// TIA Portal V18 export
ORGANIZATION_BLOCK "Main"   // OB1, LAD, ProgramCycle
TITLE = "Main Program Sweep (Cycle)"
{ S7_Optimized_Access := 'TRUE' }
VERSION : 0.1
// stored: AutoNumber true, IsIECCheckEnabled false, SetENOAutomatically false
   VAR_INPUT
      Initial_Call : Bool;   // Initial call of this OB
      Remanence : Bool;   // =True, if remanent data are available
   END_VAR
   VAR_TEMP
      temp1 : Bool;
      temp2 : Bool;
      temp3 : Bool;
      temp4 : Bool;
   END_VAR
   VAR_TEMP   // added for the SCL form of the ladder/FBD networks
      _w1 : Bool;
      _w2 : Bool;
      _w3 : Bool;
      _w4 : Bool;
      _w5 : Bool;
      _w6 : Bool;
      _w7 : Bool;
      _w8 : Bool;
      _w9 : Bool;
      _w10 : Bool;
      _w11 : Bool;
      _w12 : Bool;
      _w13 : Bool;
      _w14 : Bool;
      _w15 : Bool;
      _w16 : Bool;
   END_VAR
BEGIN

REGION Network 1: SFC1
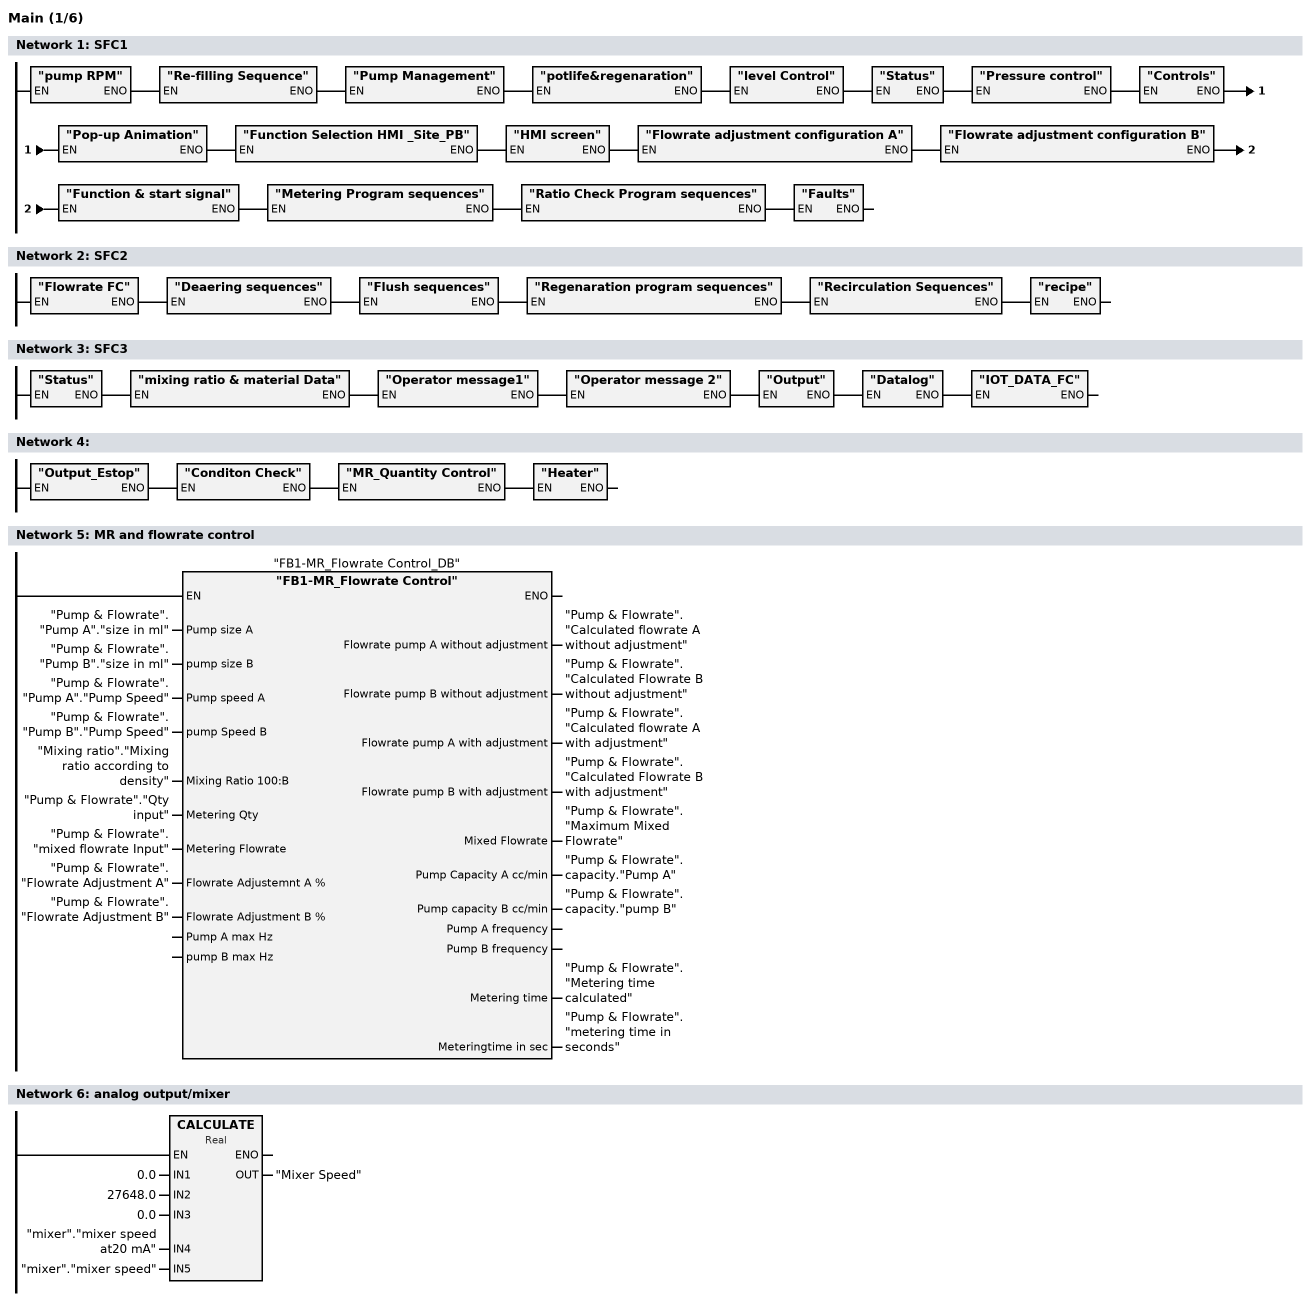
   RUNG wire#powerrail
      "pump RPM"()
      "Re-filling Sequence"()
      "Pump Management"()
      "potlife&regenaration"()
      "level Control"()
      "Status"()
      "Pressure control"()
      "Controls"()
      "Pop-up Animation"()
      "Function Selection HMI _Site_PB"()
      "HMI screen"()
      "Flowrate adjustment configuration A"()
      "Flowrate adjustment configuration B"()
      "Function & start signal"()
      "Metering Program sequences"()
      "Ratio Check Program sequences"()
      "Faults"()
   END_RUNG
   // the same network as SCL:
   "pump RPM"(ENO => #_w1);
   "Re-filling Sequence"(EN := #_w1, ENO => #_w2);
   "Pump Management"(EN := #_w2, ENO => #_w3);
   "potlife&regenaration"(EN := #_w3, ENO => #_w4);
   "level Control"(EN := #_w4, ENO => #_w5);
   "Status"(EN := #_w5, ENO => #_w6);
   "Pressure control"(EN := #_w6, ENO => #_w7);
   "Controls"(EN := #_w7, ENO => #_w8);
   "Pop-up Animation"(EN := #_w8, ENO => #_w9);
   "Function Selection HMI _Site_PB"(EN := #_w9, ENO => #_w10);
   "HMI screen"(EN := #_w10, ENO => #_w11);
   "Flowrate adjustment configuration A"(EN := #_w11, ENO => #_w12);
   "Flowrate adjustment configuration B"(EN := #_w12, ENO => #_w13);
   "Function & start signal"(EN := #_w13, ENO => #_w14);
   "Metering Program sequences"(EN := #_w14, ENO => #_w15);
   "Ratio Check Program sequences"(EN := #_w15, ENO => #_w16);
   IF #_w16 THEN "Faults"(); END_IF;
END_REGION

REGION Network 2: SFC2
   RUNG wire#powerrail
      "Flowrate FC"()
      "Deaering sequences"()
      "Flush sequences"()
      "Regenaration program sequences"()
      "Recirculation Sequences"()
      "recipe"()
   END_RUNG
   // the same network as SCL:
   "Flowrate FC"(ENO => #_w1);
   "Deaering sequences"(EN := #_w1, ENO => #_w2);
   "Flush sequences"(EN := #_w2, ENO => #_w3);
   "Regenaration program sequences"(EN := #_w3, ENO => #_w4);
   "Recirculation Sequences"(EN := #_w4, ENO => #_w5);
   IF #_w5 THEN "recipe"(); END_IF;
END_REGION

REGION Network 3: SFC3
   RUNG wire#powerrail
      "Status"()
      "mixing ratio & material Data"()
      "Operator message1"()
      "Operator message 2"()
      "Output"()
      "Datalog"()
      "IOT_DATA_FC"()
   END_RUNG
   // the same network as SCL:
   "Status"(ENO => #_w1);
   "mixing ratio & material Data"(EN := #_w1, ENO => #_w2);
   "Operator message1"(EN := #_w2, ENO => #_w3);
   "Operator message 2"(EN := #_w3, ENO => #_w4);
   "Output"(EN := #_w4, ENO => #_w5);
   "Datalog"(EN := #_w5, ENO => #_w6);
   IF #_w6 THEN "IOT_DATA_FC"(); END_IF;
END_REGION

REGION Network 4
   RUNG wire#powerrail
      "Output_Estop"()
      "Conditon Check"()
      "MR_Quantity Control"()
      "Heater"()
   END_RUNG
   // the same network as SCL:
   "Output_Estop"(ENO => #_w1);
   "Conditon Check"(EN := #_w1, ENO => #_w2);
   "MR_Quantity Control"(EN := #_w2, ENO => #_w3);
   IF #_w3 THEN "Heater"(); END_IF;
END_REGION

REGION Network 5: MR and flowrate control
   "FB1-MR_Flowrate Control_DB"("Pump size A" := "Pump & Flowrate"."Pump A"."size in ml",   // "FB1-MR_Flowrate Control"
                           "pump size B" := "Pump & Flowrate"."Pump B"."size in ml",
                           "Pump speed A" := "Pump & Flowrate"."Pump A"."Pump Speed",
                           "pump Speed B" := "Pump & Flowrate"."Pump B"."Pump Speed",
                           "Mixing Ratio 100:B" := "Mixing ratio"."Mixing ratio according to density",
                           "Metering Qty" := "Pump & Flowrate"."Qty input",
                           "Metering Flowrate" := "Pump & Flowrate"."mixed flowrate Input",
                           "Flowrate Adjustemnt A %" := "Pump & Flowrate"."Flowrate Adjustment A",
                           "Flowrate Adjustment B %" := "Pump & Flowrate"."Flowrate Adjustment B",
                           "Flowrate pump A without adjustment" => "Pump & Flowrate"."Calculated flowrate A without adjustment",
                           "Flowrate pump B without adjustment" => "Pump & Flowrate"."Calculated Flowrate B without adjustment",
                           "Flowrate pump A with adjustment" => "Pump & Flowrate"."Calculated flowrate A with adjustment",
                           "Flowrate pump B with adjustment" => "Pump & Flowrate"."Calculated Flowrate B  with adjustment",
                           "Mixed Flowrate" => "Pump & Flowrate"."Maximum Mixed Flowrate",
                           "Pump Capacity A cc/min" => "Pump & Flowrate".capacity."Pump A",
                           "Pump capacity B cc/min" => "Pump & Flowrate".capacity."pump B",
                           "Metering time" => "Pump & Flowrate"."Metering time calculated",
                           "Meteringtime in sec" => "Pump & Flowrate"."metering time in seconds");
END_REGION

REGION Network 6: analog output/mixer
   RUNG wire#powerrail
      { S7_Templates := "SrcType := Real"; S7_Expression := "(IN2-IN1)*(IN5-IN3)/(IN4-IN3)+IN1" } Calculate(in1 := 0.0, in2 := 27648.0, in3 := 0.0, in4 := "mixer"."mixer speed at20 mA", in5 := "mixer"."mixer speed", out => "Mixer Speed")
   END_RUNG
   // the same network as SCL:
   "Mixer Speed" := (27648.0-0.0)*("mixer"."mixer speed"-0.0)/("mixer"."mixer speed at20 mA"-0.0)+0.0;
END_REGION

REGION Network 7: Pump A Analog output without PID
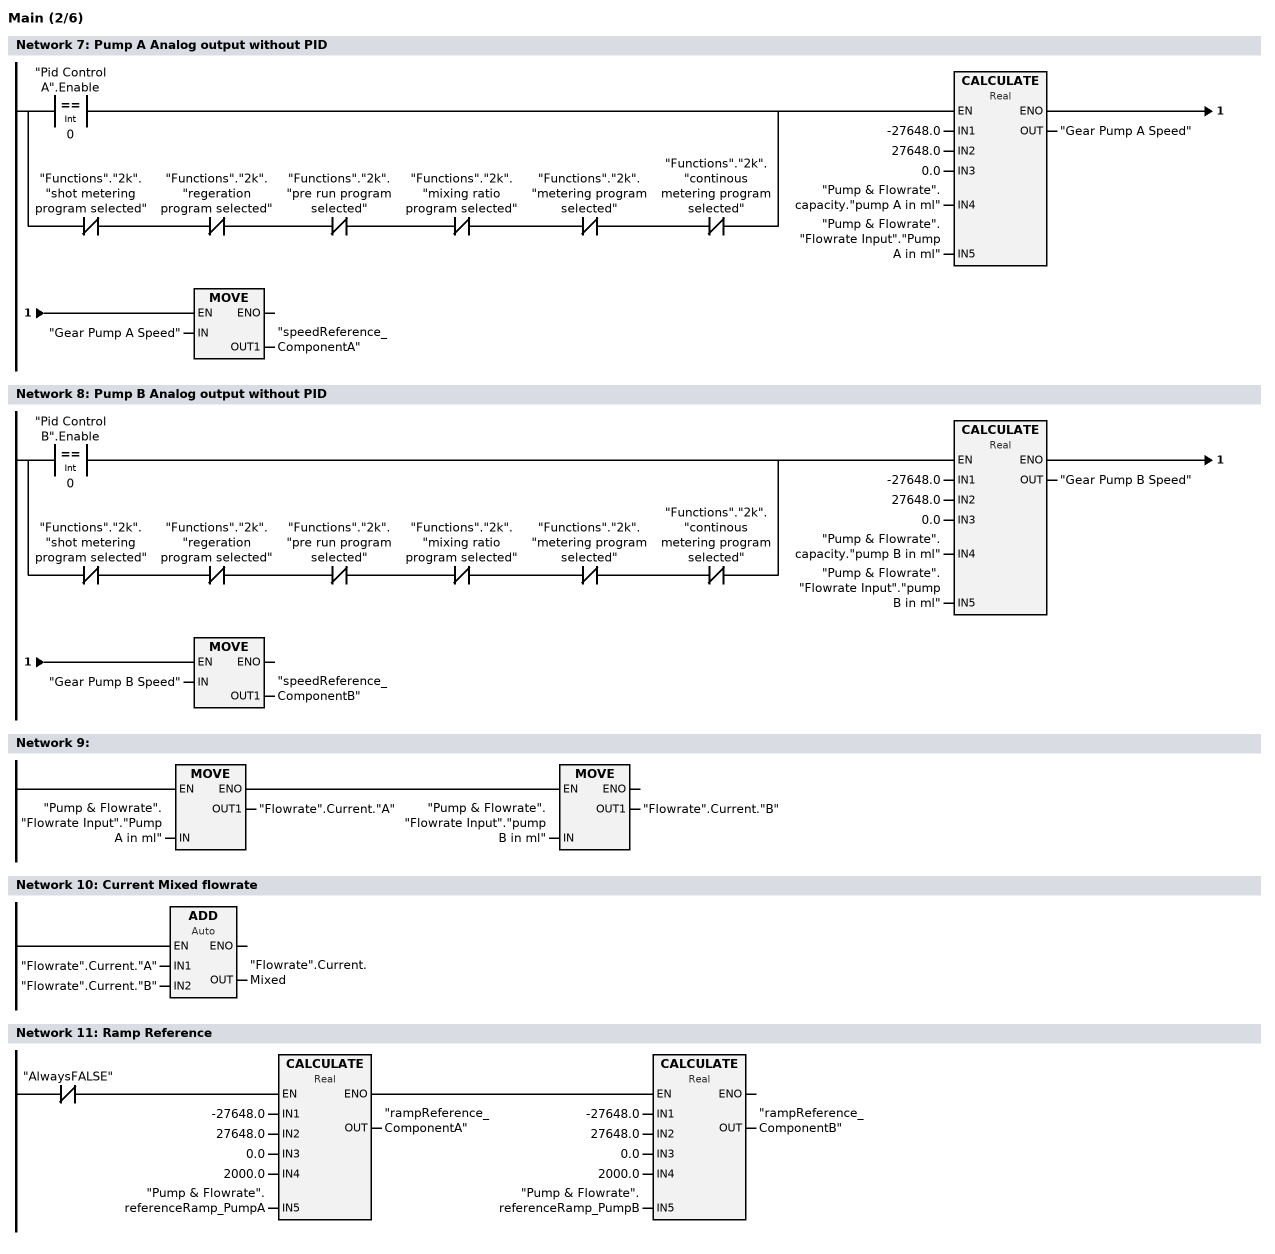
   RUNG wire#powerrail
      { S7_Templates := "SrcType := Int" } EQ_Contact(in1 := "Pid Control A".Enable, in2 := 0)
      wire#w1
      { S7_Templates := "SrcType := Real"; S7_Expression := "(IN2-IN1)*(IN5-IN3)/(IN4-IN3)+IN1" } Calculate(in1 := -27648.0, in2 := 27648.0, in3 := 0.0, in4 := "Pump & Flowrate".capacity."pump A in ml", in5 := "Pump & Flowrate"."Flowrate Input"."Pump A in ml", out => "Gear Pump A Speed")
      Move(in := "Gear Pump A Speed", out1 => "speedReference_ComponentA")
   END_RUNG
   RUNG wire#powerrail
      I_Contact( "Functions"."2k"."shot metering program selected" )
      I_Contact( "Functions"."2k"."regeration program selected" )
      I_Contact( "Functions"."2k"."pre run program selected" )
      I_Contact( "Functions"."2k"."mixing ratio program selected" )
      I_Contact( "Functions"."2k"."metering program selected" )
      I_Contact( "Functions"."2k"."continous metering program selected" )
   END_RUNG wire#w1
   // the same network as SCL:
   IF ("Pid Control A".Enable = 0) OR (NOT "Functions"."2k"."shot metering program selected" AND NOT "Functions"."2k"."regeration program selected" AND NOT "Functions"."2k"."pre run program selected" AND NOT "Functions"."2k"."mixing ratio program selected" AND NOT "Functions"."2k"."metering program selected" AND NOT "Functions"."2k"."continous metering program selected") THEN
       "Gear Pump A Speed" := (27648.0-(-27648.0))*("Pump & Flowrate"."Flowrate Input"."Pump A in ml"-0.0)/("Pump & Flowrate".capacity."pump A in ml"-0.0)+(-27648.0);
       "speedReference_ComponentA" := "Gear Pump A Speed";
   END_IF;
END_REGION

REGION Network 8: Pump B Analog output without PID
   RUNG wire#powerrail
      { S7_Templates := "SrcType := Int" } EQ_Contact(in1 := "Pid Control B".Enable, in2 := 0)
      wire#w1
      { S7_Templates := "SrcType := Real"; S7_Expression := "(IN2-IN1)*(IN5-IN3)/(IN4-IN3)+IN1" } Calculate(in1 := -27648.0, in2 := 27648.0, in3 := 0.0, in4 := "Pump & Flowrate".capacity."pump B in ml", in5 := "Pump & Flowrate"."Flowrate Input"."pump B in ml", out => "Gear Pump B Speed")
      Move(in := "Gear Pump B Speed", out1 => "speedReference_ComponentB")
   END_RUNG
   RUNG wire#powerrail
      I_Contact( "Functions"."2k"."shot metering program selected" )
      I_Contact( "Functions"."2k"."regeration program selected" )
      I_Contact( "Functions"."2k"."pre run program selected" )
      I_Contact( "Functions"."2k"."mixing ratio program selected" )
      I_Contact( "Functions"."2k"."metering program selected" )
      I_Contact( "Functions"."2k"."continous metering program selected" )
   END_RUNG wire#w1
   // the same network as SCL:
   IF ("Pid Control B".Enable = 0) OR (NOT "Functions"."2k"."shot metering program selected" AND NOT "Functions"."2k"."regeration program selected" AND NOT "Functions"."2k"."pre run program selected" AND NOT "Functions"."2k"."mixing ratio program selected" AND NOT "Functions"."2k"."metering program selected" AND NOT "Functions"."2k"."continous metering program selected") THEN
       "Gear Pump B Speed" := (27648.0-(-27648.0))*("Pump & Flowrate"."Flowrate Input"."pump B in ml"-0.0)/("Pump & Flowrate".capacity."pump B in ml"-0.0)+(-27648.0);
       "speedReference_ComponentB" := "Gear Pump B Speed";
   END_IF;
END_REGION

REGION Network 9
   RUNG wire#powerrail
      Move(in := "Pump & Flowrate"."Flowrate Input"."Pump A in ml", out1 => "Flowrate".Current."A")
      Move(in := "Pump & Flowrate"."Flowrate Input"."pump B in ml", out1 => "Flowrate".Current."B")
   END_RUNG
   // the same network as SCL:
   "Flowrate".Current."A" := "Pump & Flowrate"."Flowrate Input"."Pump A in ml";
   "Flowrate".Current."B" := "Pump & Flowrate"."Flowrate Input"."pump B in ml";
END_REGION

REGION Network 10: Current Mixed flowrate
   RUNG wire#powerrail
      Add(in1 := "Flowrate".Current."A", in2 := "Flowrate".Current."B", out => "Flowrate".Current.Mixed)
   END_RUNG
   // the same network as SCL:
   "Flowrate".Current.Mixed := "Flowrate".Current."A" + "Flowrate".Current."B";
END_REGION

REGION Network 11: Ramp Reference
   RUNG wire#powerrail
      I_Contact( "AlwaysFALSE" )
      { S7_Templates := "SrcType := Real"; S7_Expression := "ROUND((IN2-IN1)*(IN5-IN3)/(IN4-IN3)+IN1)" } Calculate(in1 := -27648.0, in2 := 27648.0, in3 := 0.0, in4 := 2000.0, in5 := "Pump & Flowrate".referenceRamp_PumpA, out => "rampReference_ComponentA")
      { S7_Templates := "SrcType := Real"; S7_Expression := "(IN2-IN1)*(IN5-IN3)/(IN4-IN3)+IN1" } Calculate(in1 := -27648.0, in2 := 27648.0, in3 := 0.0, in4 := 2000.0, in5 := "Pump & Flowrate".referenceRamp_PumpB, out => "rampReference_ComponentB")
   END_RUNG
   // the same network as SCL:
   IF NOT "AlwaysFALSE" THEN
       "rampReference_ComponentA" := ROUND((27648.0-(-27648.0))*("Pump & Flowrate".referenceRamp_PumpA-0.0)/(2000.0-0.0)+(-27648.0));
       "rampReference_ComponentB" := (27648.0-(-27648.0))*("Pump & Flowrate".referenceRamp_PumpB-0.0)/(2000.0-0.0)+(-27648.0);
   END_IF;
END_REGION

REGION Network 12: 2k Dosing running
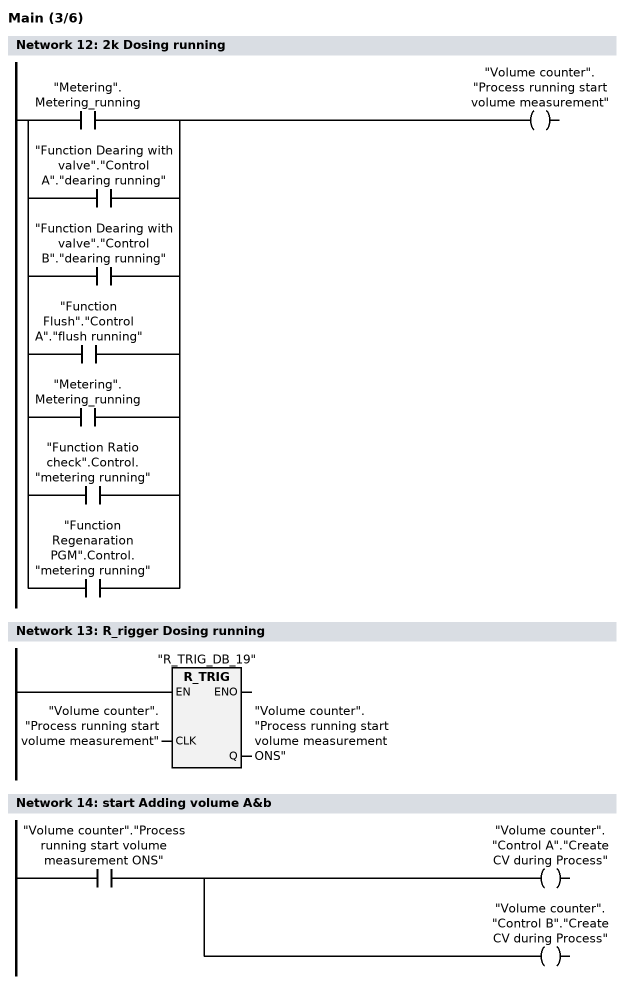
   RUNG wire#powerrail
      Contact( "Metering".Metering_running )
      wire#w1
      Coil( "Volume counter"."Process running start volume measurement" )
   END_RUNG
   RUNG wire#powerrail
      Contact( "Function Dearing with valve"."Control A"."dearing running" )
   END_RUNG wire#w1
   RUNG wire#powerrail
      Contact( "Function Dearing with valve"."Control B"."dearing running" )
   END_RUNG wire#w1
   RUNG wire#powerrail
      Contact( "Function Flush"."Control A"."flush running" )
   END_RUNG wire#w1
   RUNG wire#powerrail
      Contact( "Metering".Metering_running )
   END_RUNG wire#w1
   RUNG wire#powerrail
      Contact( "Function Ratio check".Control."metering running" )
   END_RUNG wire#w1
   RUNG wire#powerrail
      Contact( "Function Regenaration PGM".Control."metering running" )
   END_RUNG wire#w1
   // the same network as SCL:
   "Volume counter"."Process running start volume measurement" := "Metering".Metering_running OR "Function Dearing with valve"."Control A"."dearing running" OR "Function Dearing with valve"."Control B"."dearing running" OR "Function Flush"."Control A"."flush running" OR "Metering".Metering_running OR "Function Ratio check".Control."metering running" OR "Function Regenaration PGM".Control."metering running";
END_REGION

REGION Network 13: R_rigger Dosing running
   RUNG wire#powerrail
      "R_TRIG_DB_19".R_TRIG(CLK := "Volume counter"."Process running start volume measurement", Q => "Volume counter"."Process running start volume measurement ONS")
   END_RUNG
   // the same network as SCL:
   "R_TRIG_DB_19"(CLK := "Volume counter"."Process running start volume measurement",   // R_TRIG
                  Q => "Volume counter"."Process running start volume measurement ONS");
END_REGION

REGION Network 14: start Adding volume A&b
   RUNG wire#powerrail
      Contact( "Volume counter"."Process running start volume measurement ONS" )
      wire#w1
      Coil( "Volume counter"."Control A"."Create CV during Process" )
   END_RUNG
   RUNG wire#w1
      Coil( "Volume counter"."Control B"."Create CV during Process" )
   END_RUNG
   // the same network as SCL:
   "Volume counter"."Control A"."Create CV during Process" := "Volume counter"."Process running start volume measurement ONS";
   "Volume counter"."Control B"."Create CV during Process" := "Volume counter"."Process running start volume measurement ONS";
END_REGION

REGION Network 15: A volume During Operation
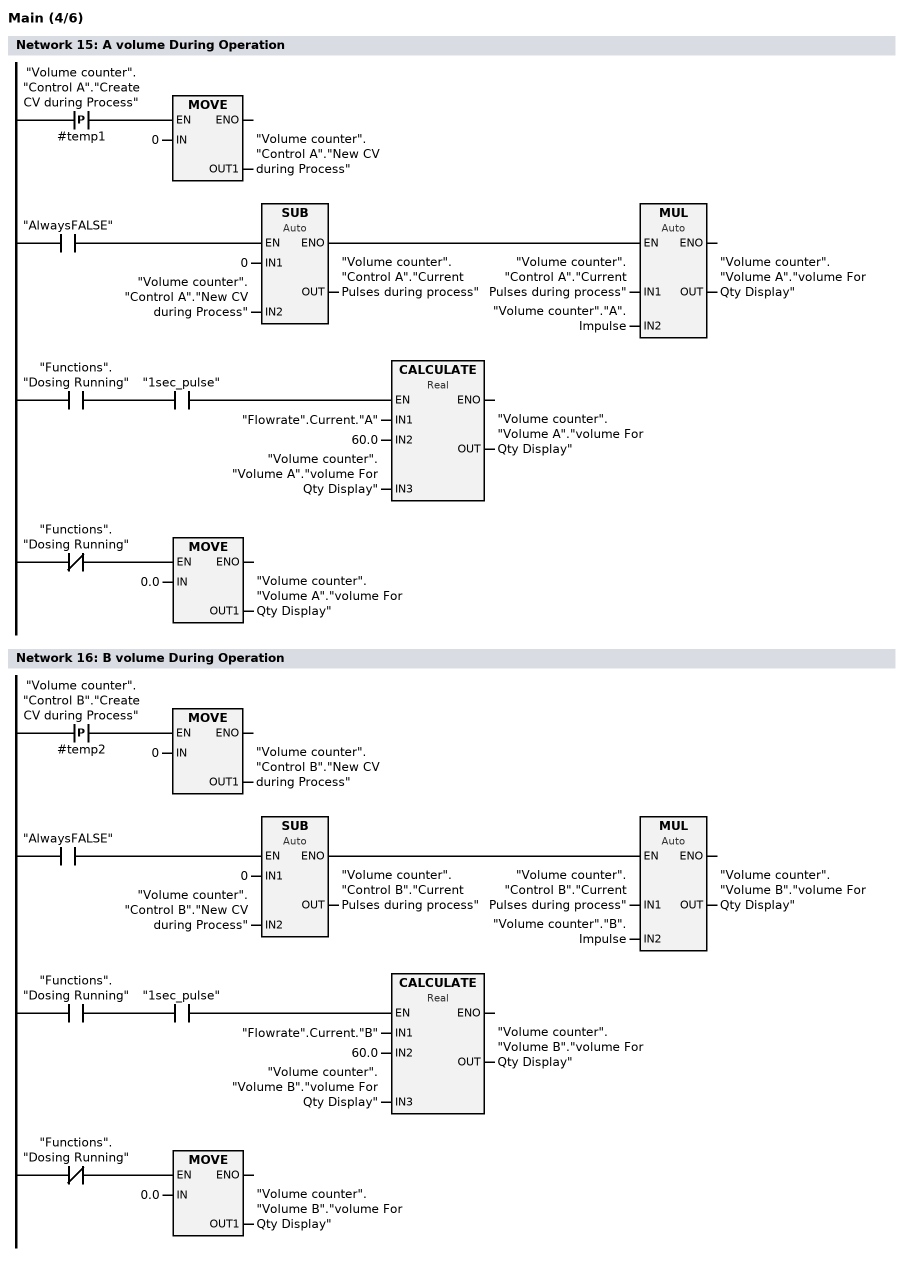
   RUNG wire#powerrail
      P_Contact(operand := "Volume counter"."Control A"."Create CV during Process", bit := #temp1)
      Move(in := 0, out1 => "Volume counter"."Control A"."New CV during Process")
   END_RUNG
   RUNG wire#powerrail
      Contact( "AlwaysFALSE" )
      Sub(in1 := 0, in2 := "Volume counter"."Control A"."New CV during Process", out => "Volume counter"."Control A"."Current Pulses during process")
      Mul(in1 := "Volume counter"."Control A"."Current Pulses during process", in2 := "Volume counter"."A".Impulse, out => "Volume counter"."Volume A"."volume For Qty Display")
   END_RUNG
   RUNG wire#powerrail
      Contact( "Functions"."Dosing Running" )
      Contact( "1sec_pulse" )
      { S7_Templates := "SrcType := Real"; S7_Expression := "(IN1/IN2)+IN3" } Calculate(in1 := "Flowrate".Current."A", in2 := 60.0, in3 := "Volume counter"."Volume A"."volume For Qty Display", out => "Volume counter"."Volume A"."volume For Qty Display")
   END_RUNG
   RUNG wire#powerrail
      I_Contact( "Functions"."Dosing Running" )
      Move(in := 0.0, out1 => "Volume counter"."Volume A"."volume For Qty Display")
   END_RUNG
   // the same network as SCL:
   #_w1 := "Volume counter"."Control A"."Create CV during Process" AND NOT #temp1;   // rising edge of "Volume counter"."Control A"."Create CV during Process"
   #temp1 := "Volume counter"."Control A"."Create CV during Process";
   IF #_w1 THEN "Volume counter"."Control A"."New CV during Process" := 0; END_IF;
   IF "AlwaysFALSE" THEN
       "Volume counter"."Control A"."Current Pulses during process" := 0 - "Volume counter"."Control A"."New CV during Process";
       "Volume counter"."Volume A"."volume For Qty Display" := "Volume counter"."Control A"."Current Pulses during process" * "Volume counter"."A".Impulse;
   END_IF;
   IF "Functions"."Dosing Running" AND "1sec_pulse" THEN
       "Volume counter"."Volume A"."volume For Qty Display" := ("Flowrate".Current."A"/60.0)+"Volume counter"."Volume A"."volume For Qty Display";
   END_IF;
   IF NOT "Functions"."Dosing Running" THEN
       "Volume counter"."Volume A"."volume For Qty Display" := 0.0;
   END_IF;
END_REGION

REGION Network 16: B volume During Operation
   RUNG wire#powerrail
      P_Contact(operand := "Volume counter"."Control B"."Create CV during Process", bit := #temp2)
      Move(in := 0, out1 => "Volume counter"."Control B"."New CV during Process")
   END_RUNG
   RUNG wire#powerrail
      Contact( "AlwaysFALSE" )
      Sub(in1 := 0, in2 := "Volume counter"."Control B"."New CV during Process", out => "Volume counter"."Control B"."Current Pulses during process")
      Mul(in1 := "Volume counter"."Control B"."Current Pulses during process", in2 := "Volume counter"."B".Impulse, out => "Volume counter"."Volume B"."volume For Qty Display")
   END_RUNG
   RUNG wire#powerrail
      Contact( "Functions"."Dosing Running" )
      Contact( "1sec_pulse" )
      { S7_Templates := "SrcType := Real"; S7_Expression := "(IN1/IN2)+IN3" } Calculate(in1 := "Flowrate".Current."B", in2 := 60.0, in3 := "Volume counter"."Volume B"."volume For Qty Display", out => "Volume counter"."Volume B"."volume For Qty Display")
   END_RUNG
   RUNG wire#powerrail
      I_Contact( "Functions"."Dosing Running" )
      Move(in := 0.0, out1 => "Volume counter"."Volume B"."volume For Qty Display")
   END_RUNG
   // the same network as SCL:
   #_w1 := "Volume counter"."Control B"."Create CV during Process" AND NOT #temp2;   // rising edge of "Volume counter"."Control B"."Create CV during Process"
   #temp2 := "Volume counter"."Control B"."Create CV during Process";
   IF #_w1 THEN "Volume counter"."Control B"."New CV during Process" := 0; END_IF;
   IF "AlwaysFALSE" THEN
       "Volume counter"."Control B"."Current Pulses during process" := 0 - "Volume counter"."Control B"."New CV during Process";
       "Volume counter"."Volume B"."volume For Qty Display" := "Volume counter"."Control B"."Current Pulses during process" * "Volume counter"."B".Impulse;
   END_IF;
   IF "Functions"."Dosing Running" AND "1sec_pulse" THEN
       "Volume counter"."Volume B"."volume For Qty Display" := ("Flowrate".Current."B"/60.0)+"Volume counter"."Volume B"."volume For Qty Display";
   END_IF;
   IF NOT "Functions"."Dosing Running" THEN
       "Volume counter"."Volume B"."volume For Qty Display" := 0.0;
   END_IF;
END_REGION

REGION Network 17: Mixed Volume During Operation
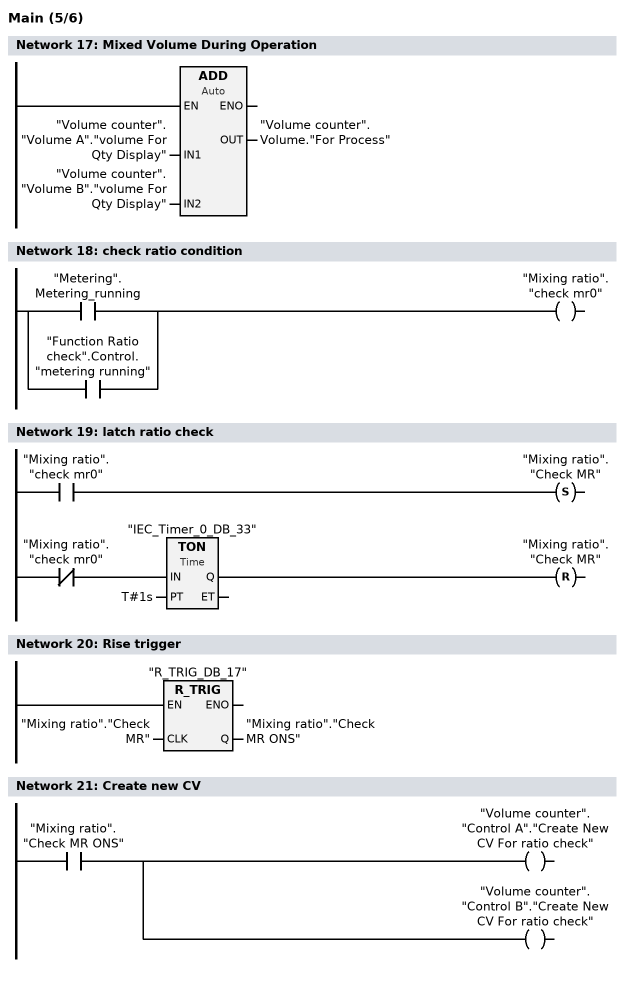
   RUNG wire#powerrail
      Add(in1 := "Volume counter"."Volume A"."volume For Qty Display", in2 := "Volume counter"."Volume B"."volume For Qty Display", out => "Volume counter".Volume."For Process")
   END_RUNG
   // the same network as SCL:
   "Volume counter".Volume."For Process" := "Volume counter"."Volume A"."volume For Qty Display" + "Volume counter"."Volume B"."volume For Qty Display";
END_REGION

REGION Network 18: check ratio condition
   RUNG wire#powerrail
      Contact( "Metering".Metering_running )
      wire#w1
      Coil( "Mixing ratio"."check mr0" )
   END_RUNG
   RUNG wire#powerrail
      Contact( "Function Ratio check".Control."metering running" )
   END_RUNG wire#w1
   // the same network as SCL:
   "Mixing ratio"."check mr0" := "Metering".Metering_running OR "Function Ratio check".Control."metering running";
END_REGION

REGION Network 19: latch ratio check
   RUNG wire#powerrail
      Contact( "Mixing ratio"."check mr0" )
      S_Coil( "Mixing ratio"."Check MR" )
   END_RUNG
   RUNG wire#powerrail
      I_Contact( "Mixing ratio"."check mr0" )
      { S7_Templates := "time_type := Time" } "IEC_Timer_0_DB_33".TON(pt := T#1s, et =>)
      R_Coil( "Mixing ratio"."Check MR" )
   END_RUNG
   // the same network as SCL:
   IF "Mixing ratio"."check mr0" THEN "Mixing ratio"."Check MR" := TRUE; END_IF;
   "IEC_Timer_0_DB_33".TON(IN := NOT "Mixing ratio"."check mr0", PT := T#1s);
   IF "IEC_Timer_0_DB_33".Q THEN "Mixing ratio"."Check MR" := FALSE; END_IF;
END_REGION

REGION Network 20: Rise trigger
   RUNG wire#powerrail
      "R_TRIG_DB_17".R_TRIG(CLK := "Mixing ratio"."Check MR", Q => "Mixing ratio"."Check MR ONS")
   END_RUNG
   // the same network as SCL:
   "R_TRIG_DB_17"(CLK := "Mixing ratio"."Check MR", Q => "Mixing ratio"."Check MR ONS");   // R_TRIG
END_REGION

REGION Network 21: Create new CV
   RUNG wire#powerrail
      Contact( "Mixing ratio"."Check MR ONS" )
      wire#w1
      Coil( "Volume counter"."Control A"."Create New CV For ratio check" )
   END_RUNG
   RUNG wire#w1
      Coil( "Volume counter"."Control B"."Create New CV For ratio check" )
   END_RUNG
   // the same network as SCL:
   "Volume counter"."Control A"."Create New CV For ratio check" := "Mixing ratio"."Check MR ONS";
   "Volume counter"."Control B"."Create New CV For ratio check" := "Mixing ratio"."Check MR ONS";
END_REGION

REGION Network 22: A volume During ratio check
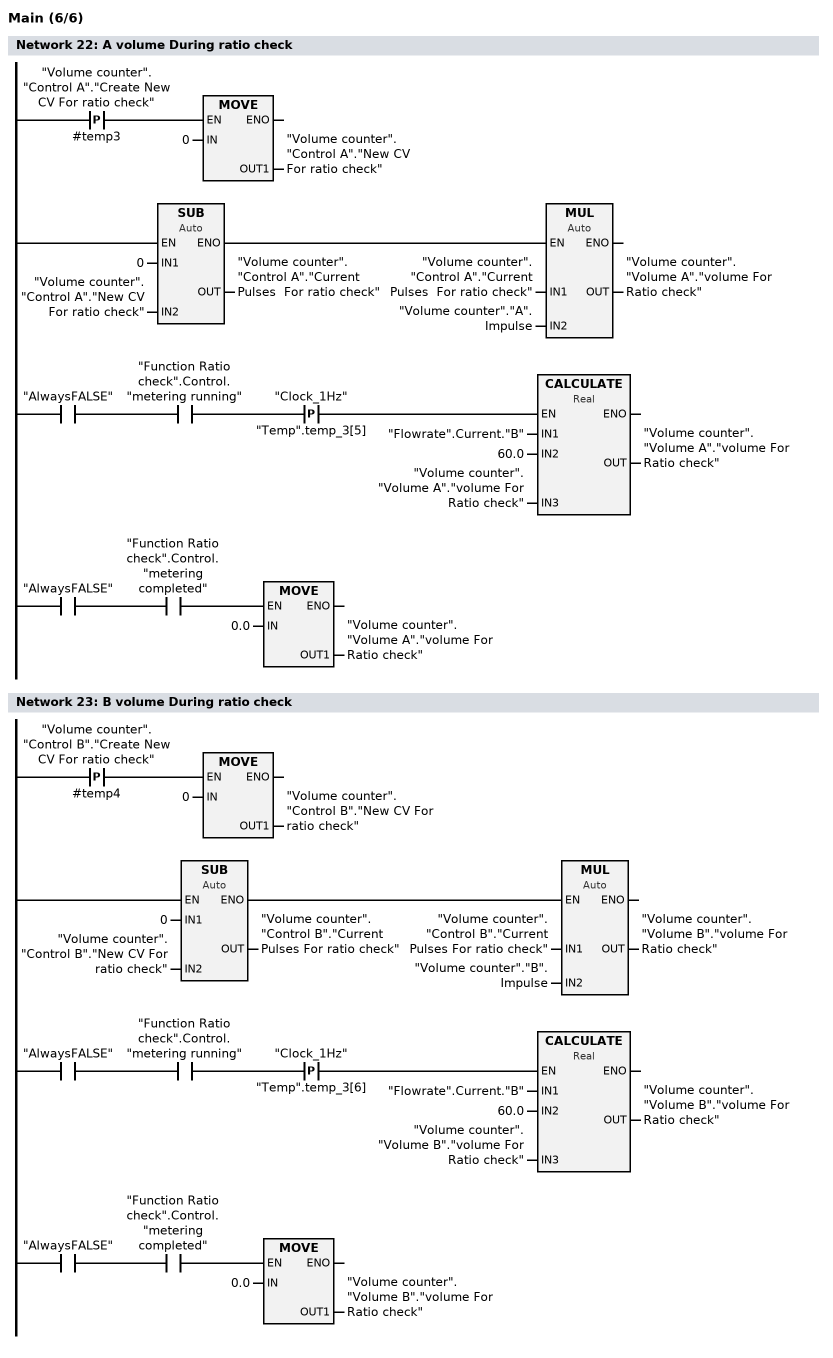
   RUNG wire#powerrail
      P_Contact(operand := "Volume counter"."Control A"."Create New CV For ratio check", bit := #temp3)
      Move(in := 0, out1 => "Volume counter"."Control A"."New CV  For ratio check")
   END_RUNG
   RUNG wire#powerrail
      Sub(in1 := 0, in2 := "Volume counter"."Control A"."New CV  For ratio check", out => "Volume counter"."Control A"."Current Pulses  For ratio check")
      Mul(in1 := "Volume counter"."Control A"."Current Pulses  For ratio check", in2 := "Volume counter"."A".Impulse, out => "Volume counter"."Volume A"."volume For Ratio check")
   END_RUNG
   RUNG wire#powerrail
      Contact( "AlwaysFALSE" )
      Contact( "Function Ratio check".Control."metering running" )
      P_Contact(operand := "Clock_1Hz", bit := "Temp".temp_3[5])
      { S7_Templates := "SrcType := Real"; S7_Expression := "(IN1/IN2)+IN3" } Calculate(in1 := "Flowrate".Current."B", in2 := 60.0, in3 := "Volume counter"."Volume A"."volume For Ratio check", out => "Volume counter"."Volume A"."volume For Ratio check")
   END_RUNG
   RUNG wire#powerrail
      Contact( "AlwaysFALSE" )
      Contact( "Function Ratio check".Control."metering completed" )
      Move(in := 0.0, out1 => "Volume counter"."Volume A"."volume For Ratio check")
   END_RUNG
   // the same network as SCL:
   #_w1 := "Volume counter"."Control A"."Create New CV For ratio check" AND NOT #temp3;   // rising edge of "Volume counter"."Control A"."Create New CV For ratio check"
   #temp3 := "Volume counter"."Control A"."Create New CV For ratio check";
   IF #_w1 THEN "Volume counter"."Control A"."New CV  For ratio check" := 0; END_IF;
   "Volume counter"."Control A"."Current Pulses  For ratio check" := 0 - "Volume counter"."Control A"."New CV  For ratio check";
   "Volume counter"."Volume A"."volume For Ratio check" := "Volume counter"."Control A"."Current Pulses  For ratio check" * "Volume counter"."A".Impulse;
   #_w2 := "AlwaysFALSE" AND "Function Ratio check".Control."metering running" AND "Clock_1Hz" AND NOT "Temp".temp_3[5];   // rising edge of "Clock_1Hz"
   "Temp".temp_3[5] := "Clock_1Hz";
   IF #_w2 THEN
       "Volume counter"."Volume A"."volume For Ratio check" := ("Flowrate".Current."B"/60.0)+"Volume counter"."Volume A"."volume For Ratio check";
   END_IF;
   IF "AlwaysFALSE" AND "Function Ratio check".Control."metering completed" THEN
       "Volume counter"."Volume A"."volume For Ratio check" := 0.0;
   END_IF;
END_REGION

REGION Network 23: B volume During ratio check
   RUNG wire#powerrail
      P_Contact(operand := "Volume counter"."Control B"."Create New CV For ratio check", bit := #temp4)
      Move(in := 0, out1 => "Volume counter"."Control B"."New CV For ratio check")
   END_RUNG
   RUNG wire#powerrail
      Sub(in1 := 0, in2 := "Volume counter"."Control B"."New CV For ratio check", out => "Volume counter"."Control B"."Current Pulses For ratio check")
      Mul(in1 := "Volume counter"."Control B"."Current Pulses For ratio check", in2 := "Volume counter"."B".Impulse, out => "Volume counter"."Volume B"."volume For Ratio check")
   END_RUNG
   RUNG wire#powerrail
      Contact( "AlwaysFALSE" )
      Contact( "Function Ratio check".Control."metering running" )
      P_Contact(operand := "Clock_1Hz", bit := "Temp".temp_3[6])
      { S7_Templates := "SrcType := Real"; S7_Expression := "(IN1/IN2)+IN3" } Calculate(in1 := "Flowrate".Current."B", in2 := 60.0, in3 := "Volume counter"."Volume B"."volume For Ratio check", out => "Volume counter"."Volume B"."volume For Ratio check")
   END_RUNG
   RUNG wire#powerrail
      Contact( "AlwaysFALSE" )
      Contact( "Function Ratio check".Control."metering completed" )
      Move(in := 0.0, out1 => "Volume counter"."Volume B"."volume For Ratio check")
   END_RUNG
   // the same network as SCL:
   #_w1 := "Volume counter"."Control B"."Create New CV For ratio check" AND NOT #temp4;   // rising edge of "Volume counter"."Control B"."Create New CV For ratio check"
   #temp4 := "Volume counter"."Control B"."Create New CV For ratio check";
   IF #_w1 THEN "Volume counter"."Control B"."New CV For ratio check" := 0; END_IF;
   "Volume counter"."Control B"."Current Pulses For ratio check" := 0 - "Volume counter"."Control B"."New CV For ratio check";
   "Volume counter"."Volume B"."volume For Ratio check" := "Volume counter"."Control B"."Current Pulses For ratio check" * "Volume counter"."B".Impulse;
   #_w2 := "AlwaysFALSE" AND "Function Ratio check".Control."metering running" AND "Clock_1Hz" AND NOT "Temp".temp_3[6];   // rising edge of "Clock_1Hz"
   "Temp".temp_3[6] := "Clock_1Hz";
   IF #_w2 THEN
       "Volume counter"."Volume B"."volume For Ratio check" := ("Flowrate".Current."B"/60.0)+"Volume counter"."Volume B"."volume For Ratio check";
   END_IF;
   IF "AlwaysFALSE" AND "Function Ratio check".Control."metering completed" THEN
       "Volume counter"."Volume B"."volume For Ratio check" := 0.0;
   END_IF;
END_REGION
END_ORGANIZATION_BLOCK
